// Implicitly generated code : DO NOT EDIT
FUNCTION CheckDivLInt : LINT
VAR_INPUT
	divisor:LINT;
END_VAR

// Implicitly generated code : Only an Implementation suggestion
{noflow}
IF divisor = 0 THEN
	CheckDivLInt:=1;
	G_Diag.uiCheckDivLint:=G_Diag.uiCheckDivLint+1;
ELSE
	CheckDivLInt:=divisor;
END_IF;
{flow}

END_FUNCTION

(* stored: Version 1.1.0.1, ProductVersion 3.1.4024.4
   POU CheckDivLInt: Id {b31ff818-cfa0-4e51-aeda-d06ee57ae2a7}, SpecialFunc CheckDivInt64 *)
